Fanuc KAREL source: kb00133.KL

-- PROVISIONAL review KL for V1013-1; original PC SHA256 5241c9094357b7732326f188100d6df8360c8ba2a1f7cda34c32e65d7a69f095
-- Incomplete behavior may be omitted. Consult companion uncertainty JSON. Do not deploy.
PROGRAM KB00133
%NOLOCKGROUP
BEGIN
  -- UNRESOLVED_PC offsets 5-12; opcodes 9D,23
  -- UNRESOLVED_PC offsets 17-24; opcodes 9D,23
  -- UNRESOLVED_PC offsets 29-36; opcodes 9D,23
  -- UNRESOLVED_PC offsets 41-48; opcodes 9D,23
  -- UNRESOLVED_PC offsets 53-60; opcodes 9D,23
  -- UNRESOLVED_PC offsets 65-99; opcodes 27,22,22,22,22,22,31
  -- UNRESOLVED_PC offsets 104-108; opcodes 7F
END KB00133
